// TwinCAT 3 PLC project ADS_lib
// Title: Ads_lib
// Company: Chua Siang Poh
// Author: Chua Siang Poh
// ProjectVersion: 1.0.0
// ProgramVersion: 3.1.4020.10
// libraries:
//   Tc2_Standard, * (Beckhoff Automation GmbH)
//   Tc2_System, * (Beckhoff Automation GmbH)
//   Tc3_Interfaces, * (Beckhoff Automation GmbH)
//   Tc3_Module, * (Beckhoff Automation GmbH)
// project tree:
//   Base Component/Class/ C_ADSCLIENT.TcPOU
// (motion and I/O tree: see PLC project motion_library)
// real-time tasks:
//   TASK PlcTask: cycle T#10ms, priority 20, ADS port 350

// ---- Base Component/Class/C_ADSCLIENT.TcPOU
FUNCTION_BLOCK C_ADSCLIENT
VAR_INPUT
END_VAR
VAR_OUTPUT
END_VAR
VAR
	_AMSID 		: STRING(23);
	_AMSPORT	: UINT := 851;	
	_TIMEOUT	: TIME := T#5S;
	
	_FBREAD		: ADSREAD;
	_FBWRITE	: ADSWRITE;
	_FBRDWRT	: ADSRDWRT;
	_FBSETCTRL	: ADSWRTCTL;
END_VAR

METHOD CREATE_HANDLE : DINT
VAR_INPUT
	VARIABLE_NAME 	: STRING(255);
	HANDLE_OUT		: POINTER TO UDINT;
END_VAR
_FBRDWRT(
	NETID:= NET_ID, 
	PORT:= PORT, 
	IDXGRP:= 16#F003, 
	IDXOFFS:= 0, 
	WRITELEN:= LEN(VARIABLE_NAME), 
	READLEN:= 4, 
	SRCADDR:= ADR(VARIABLE_NAME), 
	DESTADDR:= HANDLE_OUT, 
	WRTRD:= TRUE, 
	TMOUT:= TIMEOUT, 
	BUSY=> , 
	ERR=> , 
	ERRID=> );
IF _FBRDWRT.ERR THEN
	 _FBRDWRT( WRTRD:= FALSE );
	 CREATE_HANDLE := 1;
	 RETURN;
ELSIF NOT _FBRDWRT.BUSY THEN
	 _FBRDWRT( WRTRD:= FALSE );
	 CREATE_HANDLE := -1;
	 RETURN;
ELSE
	 CREATE_HANDLE := 0;
	 RETURN;
END_IF
END_METHOD

PROPERTY NET_ID : STRING(23)
GET
NET_ID := _AMSID;
END_GET
SET
_AMSID := NET_ID;
END_SET
END_PROPERTY

PROPERTY PORT : UINT
GET
PORT := _AMSPORT;
END_GET
SET
_AMSPORT := PORT;
END_SET
END_PROPERTY

METHOD READ_BY_HANDLE : DINT
VAR_INPUT
	HANDLE 		: UDINT;
	LENGTH 		: UDINT;
	POINTER_OUT	: PVOID;
END_VAR
_FBREAD(
	NETID:= _AMSID, 
	PORT:= _AMSPORT, 
	IDXGRP:= 16#F005, 
	IDXOFFS:= HANDLE, 
	LEN:= LENGTH, 
	DESTADDR:= POINTER_OUT, 
	READ:= TRUE, 
	TMOUT:= TIMEOUT, 
	BUSY=> , 
	ERR=> , 
	ERRID=> );
IF _FBREAD.ERR THEN
	_FBREAD( READ:= FALSE );
	READ_BY_HANDLE := 1;
	RETURN;
ELSIF NOT _FBREAD.BUSY THEN
	_FBREAD( READ:= FALSE );
	READ_BY_HANDLE := -1;
	RETURN;
ELSE
	READ_BY_HANDLE := 0;
	RETURN;
END_IF
END_METHOD

METHOD RELEASE_HANDLE : DINT
VAR_INPUT
	HANDLE : UDINT;
END_VAR
_FBWRITE(
	NETID:= NET_ID, 
	PORT:= PORT,
	IDXGRP:= 16#F006, 
	IDXOFFS:= 0, 
	LEN:= 4, 
	SRCADDR:= ADR(HANDLE), 
	WRITE:= TRUE, 
	TMOUT:= TIMEOUT, 
	BUSY=> , 
	ERR=> , 
	ERRID=> );
IF _FBWRITE.ERR THEN
	_FBWRITE( WRITE:= FALSE );
	RELEASE_HANDLE := 1;
	RETURN;
ELSIF NOT _FBWRITE.BUSY THEN
	_FBWRITE( WRITE:= FALSE );
	RELEASE_HANDLE := -1;
	RETURN;
ELSE
	RELEASE_HANDLE := 0;
	RETURN;
END_IF
END_METHOD

PROPERTY TIMEOUT : TIME
GET
TIMEOUT := _TIMEOUT;
END_GET
SET
_TIMEOUT := TIMEOUT;
END_SET
END_PROPERTY

METHOD WRITE_BY_HANDLE : DINT
VAR_INPUT
	HANDLE 		: UDINT;
	LENGTH 		: UDINT;
	POINTER_IN	: PVOID;
END_VAR
_FBWRITE(
	NETID:= _AMSID, 
	PORT:= _AMSPORT, 
	IDXGRP:= 16#F005, 
	IDXOFFS:= HANDLE,
	LEN:= LENGTH, 
	SRCADDR:= POINTER_IN, 
	WRITE:= TRUE, 
	TMOUT:= TIMEOUT, 
	BUSY=> , 
	ERR=> , 
	ERRID=> );
IF _FBWRITE.ERR THEN
	_FBWRITE( WRITE:= FALSE );
	WRITE_BY_HANDLE := 1;
	RETURN;
ELSIF NOT _FBWRITE.BUSY THEN
	_FBWRITE( WRITE:= FALSE );
	WRITE_BY_HANDLE := -1;
	RETURN;
ELSE
	WRITE_BY_HANDLE := 0;
	RETURN;
END_IF
END_METHOD

END_FUNCTION_BLOCK
